(************************************************************************************************
*
*Max pressure DO
*
***********************************************************************************************)

TYPE PMAX_DO :
STRUCT

	WAGON_WAIT_CYLINDER:BOOL;
	WAGON_LOCK_CYLINDER:BOOL;
	WAGON_STOP_CYLINDER:BOOL;
	HYDRO_CYLINDER_TOP:BOOL;
	HYDRO_CYLINDER_BOT:BOOL;
	ELECTR_CYLINDER:BOOL;
	Y7:BOOL;
	Y8:BOOL;
	PUMP_POWER:BOOL;
	PRESSURE_VALVE:BOOL;
	WATER_TANK_VALVE:BOOL;
	FLOW_STOP_VALVE:BOOL;
	FLOW_STOP_BOTT:BOOL;

END_STRUCT
END_TYPE

(* stored: Version 1.1.0.1, ProductVersion 3.1.0.26
   DUT PMAX_DO: Id {f026bab2-0497-4c90-9272-64cb0e2cdb63} *)
